Fanuc TP program (LS listing): UP021.LS

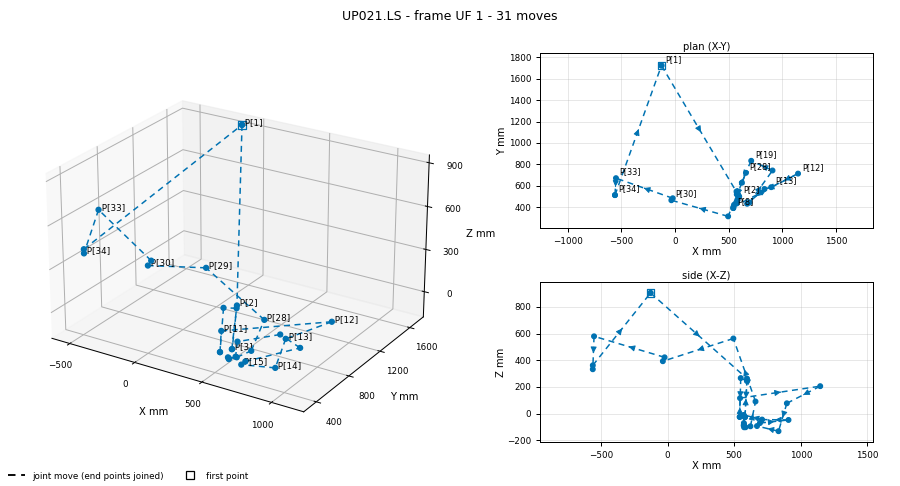
[picture p0: tool path of UP021.LS in frame UF 1, 31 of 37 moves have a stored position in this frame; points joined in program order, loops and branches not executed]
/PROG  UP021
/ATTR
OWNER		= GME;
COMMENT		= "Soldar en ST160i";
PROG_SIZE	= 14572;
CREATE		= DATE 03-01-31  TIME 09:09:48;
MODIFIED	= DATE 24-06-01  TIME 09:33:14;
FILE_NAME	= UP021;
VERSION		= 0;
LINE_COUNT	= 63;
MEMORY_SIZE	= 28492;
PROTECT		= READ_WRITE;
TCD:  STACK_SIZE	= 500,
      TASK_PRIORITY	= 50,
      TIME_SLICE	= 0,
      BUSY_LAMP_OFF	= 0,
      ABORT_REQUEST	= 0,
      PAUSE_REQUEST	= 0;
DEFAULT_GROUP	= 1,1,1,1,*;
CONTROL_CODE	= 00000000 00000000;
/APPL
/MN
   1:  UFRAME_NUM=1 ;
   2:  UTOOL_NUM=1 ;
   3:  PAYLOAD[1] ;
   4:  !Apagar Perfil Lib. 80 vs ST1600 ;
   5:  !Apagar Perfil Lib. 79 vs ST1600 ;
   6:  !Endender Anticol. 1 vs 1550R01 ;
   7:  !Endender Anticol. 3 vs 1610R01 ;
   8:J P[1] 100% CNT0 ACC100 TB    0.00sec,P-SPS    ;
      1:  TC_ONLINE (ON) ;
      2:  DO[23]=OFF ;
      3:  TIMER[3]=RESET ;
      4:  TIMER[3]=START ;
      5:  CALL MAKRO050    ;
      6:  !Lib. de Herramientas ;
      7:  DO[79]=ON ;
      8:  DO[80]=ON ;
      9:  !Lib. de Anticolisiones ;
     10:  DO[41]=ON ;
     11:  DO[42]=ON ;
     12:  DO[43]=ON ;
     13:  DO[44]=ON ;
     14:  !Apagar Pos. Base ;
     15:  DO[15]=OFF ;
     16:  !Robot en Trayectoria ;
     17:  DO[16]=ON ;
     18:  WAIT (DI[79] AND DI[80])    ;
     19:  DO[80]=OFF ;
     20:  DO[79]=OFF ;
     21:  !Encender Anticolisiones ;
     22:  DO[81]=ON ;
     23:  DO[83]=ON ;
     24:  CALL MAKRO020    ;
     25:  WAIT (DI[23])    ;
     26:  DO[23]=ON ;
     27:  TC_ONLINE (DI[41] AND DI[43] AND DI[79] AND DI[80] AND M[30] AND M[95]) ;
       ------ ;
   9:J P[2] 100% CNT100 ACC100 TB   0.00sec,P-SPS    ;
      1:  TC_ONLINE (DI[41] AND DI[43] AND DI[79] AND DI[80] AND M[30] AND M[95]) ;
       ------ ;
  10:J P[3] 100% CNT100 ACC100 TB   0.00sec,P-SPS    ;
      1:  TC_ONLINE (DI[41] AND DI[43] AND DI[79] AND DI[80] AND M[30] AND M[95]) ;
       ------ ;
  11:  !Punto de Sol. No. 11634 ;
  12:  !5qa803091b_p0008_h0210005900 ;
  13:J P[4] 100% CNT0 ACC100 TB    .10sec,P-SPS Tool_Offset,PR[11] Offset,PR[12]    ;
      1:  TC_ONLINE (ON) ;
      2:  DO[23]=OFF ;
      3:  WAIT (!DI[16] AND DI[23])    ;
      4:  CALL VW_USER(Basic1,EZSP,Nr1,ProgNr=99, , ,S-Punkt=11634,Fzg_Typ=7,EIN/AUS=ON) ;
      5:  GO[2]=(R[197]-2) ;
      6:  WAIT (!DI[129] OR DI[26])    ;
      7:  CALL MAKRO080    ;
      8:  WAIT (DI[23])    ;
      9:  DO[23]=ON ;
     10:  TC_ONLINE (DI[41] AND DI[43] AND DI[79] AND DI[80] AND M[30] AND M[95]) ;
       ------ ;
  14:J P[5] 100% CNT100 ACC100 TB   0.00sec,P-SPS    ;
      1:  TC_ONLINE (DI[41] AND DI[43] AND DI[79] AND DI[80] AND M[30] AND M[95]) ;
       ------ ;
  15:J P[6] 100% CNT100 ACC100 TB   0.00sec,P-SPS    ;
      1:  TC_ONLINE (DI[41] AND DI[43] AND DI[79] AND DI[80] AND M[30] AND M[95]) ;
       ------ ;
  16:J P[7] 100% CNT100 ACC100 TB   0.00sec,P-SPS    ;
      1:  TC_ONLINE (DI[41] AND DI[43] AND DI[79] AND DI[80] AND M[30] AND M[95]) ;
       ------ ;
  17:J P[8] 100% CNT100 ACC100 TB   0.00sec,P-SPS    ;
      1:  TC_ONLINE (DI[41] AND DI[43] AND DI[79] AND DI[80] AND M[30] AND M[95]) ;
       ------ ;
  18:  !Punto de Sol. No. 11635 ;
  19:  !5qa803091b_p0008_h0210006400 ;
  20:J P[9] 100% CNT0 ACC100 TB    .10sec,P-SPS Tool_Offset,PR[11] Offset,PR[12]    ;
      1:  TC_ONLINE (ON) ;
      2:  DO[23]=OFF ;
      3:  WAIT (!DI[16] AND DI[23])    ;
      4:  CALL VW_USER(Basic1,EZSP,Nr1,ProgNr=99, , ,S-Punkt=11635,Fzg_Typ=7,EIN/AUS=ON) ;
      5:  GO[2]=(R[197]-2) ;
      6:  WAIT (!DI[129] OR DI[26])    ;
      7:  CALL MAKRO080    ;
      8:  WAIT (DI[23])    ;
      9:  DO[23]=ON ;
     10:  TC_ONLINE (DI[41] AND DI[43] AND DI[79] AND DI[80] AND M[30] AND M[95]) ;
       ------ ;
  21:J P[10] 100% CNT100 ACC100 TB   0.00sec,P-SPS    ;
      1:  TC_ONLINE (DI[41] AND DI[43] AND DI[79] AND DI[80] AND M[30] AND M[95]) ;
       ------ ;
  22:J P[11] 100% CNT100 ACC100 TB   0.00sec,P-SPS    ;
      1:  TC_ONLINE (DI[41] AND DI[43] AND DI[79] AND DI[80] AND M[30] AND M[95]) ;
       ------ ;
  23:J P[12] 100% CNT100 ACC100 TB   0.00sec,P-SPS    ;
      1:  TC_ONLINE (DI[41] AND DI[43] AND DI[79] AND DI[80] AND M[30] AND M[95]) ;
       ------ ;
  24:J P[13] 100% CNT100 ACC100 TB   0.00sec,P-SPS    ;
      1:  TC_ONLINE (DI[41] AND DI[43] AND DI[79] AND DI[80] AND M[30] AND M[95]) ;
       ------ ;
  25:J P[14] 100% CNT100 ACC100 TB   0.00sec,P-SPS    ;
      1:  TC_ONLINE (DI[41] AND DI[43] AND DI[79] AND DI[80] AND M[30] AND M[95]) ;
       ------ ;
  26:J P[15] 100% CNT100 ACC100 TB   0.00sec,P-SPS    ;
      1:  TC_ONLINE (DI[41] AND DI[43] AND DI[79] AND DI[80] AND M[30] AND M[95]) ;
       ------ ;
  27:  !Punto de Sol. No. 11636 ;
  28:  !5qa803091b_p0008_h0210007000 ;
  29:J P[16] 100% CNT0 ACC100 TB    .10sec,P-SPS Tool_Offset,PR[11] Offset,PR[12]    ;
      1:  TC_ONLINE (ON) ;
      2:  DO[23]=OFF ;
      3:  WAIT (!DI[16] AND DI[23])    ;
      4:  CALL VW_USER(Basic1,EZSP,Nr1,ProgNr=99, , ,S-Punkt=11636,Fzg_Typ=7,EIN/AUS=ON) ;
      5:  GO[2]=(R[197]+10) ;
      6:  WAIT (!DI[129] OR DI[26])    ;
      7:  CALL MAKRO080    ;
      8:  WAIT (DI[23])    ;
      9:  DO[23]=ON ;
     10:  TC_ONLINE (DI[41] AND DI[43] AND DI[79] AND DI[80] AND M[30] AND M[95]) ;
       ------ ;
  30:J P[17] 100% CNT100 ACC100 TB   0.00sec,P-SPS    ;
      1:  TC_ONLINE (DI[41] AND DI[43] AND DI[79] AND DI[80] AND M[30] AND M[95]) ;
       ------ ;
  31:J P[18] 100% CNT100 ACC100 TB   0.00sec,P-SPS    ;
      1:  TC_ONLINE (DI[41] AND DI[43] AND DI[79] AND DI[80] AND M[30] AND M[95]) ;
       ------ ;
  32:J P[19] 100% CNT100 ACC100 TB   0.00sec,P-SPS    ;
      1:  TC_ONLINE (DI[41] AND DI[43] AND DI[79] AND DI[80] AND M[30] AND M[95]) ;
       ------ ;
  33:J P[20] 100% CNT100 ACC100 TB   0.00sec,P-SPS    ;
      1:  TC_ONLINE (DI[41] AND DI[43] AND DI[79] AND DI[80] AND M[30] AND M[95]) ;
       ------ ;
  34:J P[21] 100% CNT100 ACC100 TB   0.00sec,P-SPS    ;
      1:  TC_ONLINE (DI[41] AND DI[43] AND DI[79] AND DI[80] AND M[30] AND M[95]) ;
       ------ ;
  35:J P[22] 100% CNT100 ACC100 TB   0.00sec,P-SPS    ;
      1:  TC_ONLINE (DI[41] AND DI[43] AND DI[79] AND DI[80] AND M[30] AND M[95]) ;
       ------ ;
  36:J P[23] 100% CNT100 ACC100 TB   0.00sec,P-SPS    ;
      1:  TC_ONLINE (DI[41] AND DI[43] AND DI[79] AND DI[80] AND M[30] AND M[95]) ;
       ------ ;
  37:  !Punto de Sol. No. 11637 ;
  38:  !5qa803091b_p0008_h0210006100 ;
  39:J P[24] 100% CNT0 ACC100 TB    .10sec,P-SPS Tool_Offset,PR[11] Offset,PR[12]    ;
      1:  TC_ONLINE (ON) ;
      2:  DO[23]=OFF ;
      3:  WAIT (!DI[16] AND DI[23])    ;
      4:  CALL VW_USER(Basic1,EZSP,Nr1,ProgNr=99, , ,S-Punkt=11637,Fzg_Typ=7,EIN/AUS=ON) ;
      5:  GO[2]=(R[197]+10) ;
      6:  WAIT (!DI[129] OR DI[26])    ;
      7:  CALL MAKRO080    ;
      8:  WAIT (DI[23])    ;
      9:  DO[23]=ON ;
     10:  TC_ONLINE (DI[41] AND DI[43] AND DI[79] AND DI[80] AND M[30] AND M[95]) ;
       ------ ;
  40:J P[25] 100% CNT100 ACC100 TB   0.00sec,P-SPS    ;
      1:  TC_ONLINE (DI[41] AND DI[43] AND DI[79] AND DI[80] AND M[30] AND M[95]) ;
       ------ ;
  41:J P[26] 100% CNT100 ACC100 TB   0.00sec,P-SPS    ;
      1:  TC_ONLINE (DI[41] AND DI[43] AND DI[79] AND DI[80] AND M[30] AND M[95]) ;
       ------ ;
  42:J P[27] 100% CNT100 ACC100 TB   0.00sec,P-SPS    ;
      1:  TC_ONLINE (DI[41] AND DI[43] AND DI[79] AND DI[80] AND M[30] AND M[95]) ;
       ------ ;
  43:J P[28] 100% CNT100 ACC100 TB   0.00sec,P-SPS    ;
      1:  TC_ONLINE (DI[41] AND DI[43] AND DI[79] AND DI[80] AND M[30] AND M[95]) ;
       ------ ;
  44:J P[29] 100% CNT100 ACC100 TB   0.00sec,P-SPS    ;
      1:  TC_ONLINE (DI[41] AND DI[43] AND DI[79] AND DI[80] AND M[30] AND M[95]) ;
       ------ ;
  45:J P[30] 100% CNT100 ACC100 TB   0.00sec,P-SPS    ;
      1:  TC_ONLINE (DI[41] AND DI[43] AND DI[79] AND DI[80] AND M[30] AND M[95]) ;
       ------ ;
  46:  !no soldar CKD ;
  47:  !Punto de Sol. No. 11638 ;
  48:  !5qa802035b_018_sps0033_R ;
  49:J P[31] 100% CNT0 ACC100 TB    .10sec,P-SPS Tool_Offset,PR[11] Offset,PR[12]    ;
      1:  TC_ONLINE (ON) ;
      2:  DO[23]=OFF ;
      3:  WAIT (!DI[16] AND DI[23])    ;
      4:  CALL VW_USER(Basic1,EZSP,Nr1,ProgNr=99, , ,S-Punkt=11638,Fzg_Typ=7,EIN/AUS=ON) ;
      5:  GO[2]=(R[197]-4) ;
      6:  WAIT (!DI[129] OR DI[26])    ;
      7:  CALL MAKRO080    ;
      8:  WAIT (DI[23])    ;
      9:  DO[23]=ON ;
     10:  TC_ONLINE (DI[41] AND DI[43] AND DI[79] AND DI[80] AND M[30] AND M[95]) ;
       ------ ;
  50:J P[32] 100% CNT100 ACC100 TB   0.00sec,P-SPS    ;
      1:  TC_ONLINE (DI[41] AND DI[43] AND DI[79] AND DI[80] AND M[30] AND M[95]) ;
       ------ ;
  51:J P[33] 100% FINE ACC100 DB    0.0mm,P-SPS    ;
      1:  TC_ONLINE (DI[41] AND DI[43] AND DI[79] AND DI[80] AND M[30] AND M[95]) ;
       ------ ;
  52:J P[34] 100% CNT100 ACC100 TB   0.00sec,P-SPS    ;
      1:  TC_ONLINE (DI[41] AND DI[43] AND DI[79] AND DI[80] AND M[30] AND M[95]) ;
       ------ ;
  53:  !no soldar CKD ;
  54:  !Punto de Sol. No. 11639 ;
  55:  !Fin de Trabajo 1 ;
  56:  !5qa802035b_018_sps0021_R ;
  57:J P[35] 100% CNT0 ACC100 TB    0.00sec,P-SPS Tool_Offset,PR[11] Offset,PR[12]    ;
      1:  TC_ONLINE (ON) ;
      2:  DO[23]=OFF ;
      3:  WAIT (!DI[16] AND DI[23])    ;
      4:  CALL VW_USER(Basic1,EZSP,Nr1,ProgNr=99, , ,S-Punkt=11639,Fzg_Typ=7,EIN/AUS=ON) ;
      5:  GO[2]=(R[197]) ;
      6:  WAIT (!DI[129] OR DI[26])    ;
      7:  CALL MAKRO080    ;
      8:  IF (!DI[145] AND !DI[129]),CALL MAKRO001 ;
      9:  WAIT (DI[23])    ;
     10:  DO[23]=ON ;
     11:  TC_ONLINE (DI[41] AND DI[43] AND DI[79] AND DI[80] AND M[30] AND M[95]) ;
       ------ ;
  58:J P[36] 100% CNT100 ACC100 TB   0.00sec,P-SPS    ;
      1:  TC_ONLINE (DI[41] AND DI[43] AND DI[79] AND DI[80] AND M[30] AND M[95]) ;
       ------ ;
  59:  !Encender Perfil Lib 80 vs ST1600 ;
  60:  !Encender Perfil Lib 79 vs ST1600 ;
  61:  !Apagar Anticol. 1 vs 1550R01 ;
  62:  !Apagar Anticol. 3 vs 1610R01 ;
  63:J P[37] 100% CNT0 ACC100 TB    .10sec,P-SPS    ;
      1:  TC_ONLINE (ON) ;
      2:  DO[23]=OFF ;
      3:  TIMER[3]=STOP ;
      4:  DO[41]=ON ;
      5:  DO[43]=ON ;
      6:  DO[79]=ON ;
      7:  DO[80]=ON ;
      8:  WAIT (DI[23])    ;
      9:  DO[23]=ON ;
     10:  TC_ONLINE (M[30] AND M[95]) ;
       ------ ;
/POS
P[1]{
   GP1:
	UF : 1, UT : 1,		CONFIG : 'N U T, 0, 0, 0',
	X =  -127.542  mm,	Y =  1721.879  mm,	Z =   904.497  mm,
	W =  -170.302 deg,	P =     1.120 deg,	R =   132.757 deg
   GP2:
	UF : 1, UT : 1,
	J1=   100.000  mm
   GP3:
	UF : 1, UT : 1,
	J1=     0.000  mm
   GP4:
	UF : 1, UT : 1,
	J1=     0.000  mm
};
P[2]{
   GP1:
	UF : 1, UT : 1,		CONFIG : 'N U T, 0, 0, 0',
	X =   596.207  mm,	Y =   502.707  mm,	Z =   261.856  mm,
	W =  -176.468 deg,	P =     7.977 deg,	R =    93.412 deg
   GP2:
	UF : 1, UT : 1,
	J1=   125.000  mm
   GP3:
	UF : 1, UT : 1,
	J1=     0.000  mm
   GP4:
	UF : 1, UT : 1,
	J1=     0.000  mm
};
P[3]{
   GP1:
	UF : 1, UT : 1,		CONFIG : 'N U T, 0, 0, 0',
	X =   580.717  mm,	Y =   471.716  mm,	Z =   -27.286  mm,
	W =  -176.468 deg,	P =     7.977 deg,	R =    93.413 deg
   GP2:
	UF : 1, UT : 1,
	J1=   125.000  mm
   GP3:
	UF : 1, UT : 1,
	J1=     0.000  mm
   GP4:
	UF : 1, UT : 1,
	J1=     0.000  mm
};
P[4]{
   GP1:
	UF : 1, UT : 1,		CONFIG : 'N U T, 0, 0, 0',
	X =   579.173  mm,	Y =   480.025  mm,	Z =   -30.338  mm,
	W =  -175.927 deg,	P =     7.716 deg,	R =    97.374 deg
   GP2:
	UF : 1, UT : 1,
	J1=    14.100  mm
   GP3:
	UF : 1, UT : 1,
	J1=     0.000  mm
   GP4:
	UF : 1, UT : 1,
	J1=     0.000  mm
};
P[5]{
   GP1:
	UF : 1, UT : 1,		CONFIG : 'N U T, 0, 0, 0',
	X =   581.000  mm,	Y =   466.971  mm,	Z =   -26.620  mm,
	W =  -176.468 deg,	P =     7.977 deg,	R =    93.413 deg
   GP2:
	UF : 1, UT : 1,
	J1=   125.000  mm
   GP3:
	UF : 1, UT : 1,
	J1=     0.000  mm
   GP4:
	UF : 1, UT : 1,
	J1=     0.000  mm
};
P[6]{
   GP1:
	UF : 1, UT : 1,		CONFIG : 'N U T, 0, 0, 0',
	X =   595.238  mm,	Y =   500.117  mm,	Z =   243.816  mm,
	W =  -176.468 deg,	P =     7.977 deg,	R =    93.412 deg
   GP2:
	UF : 1, UT : 1,
	J1=   125.000  mm
   GP3:
	UF : 1, UT : 1,
	J1=     0.000  mm
   GP4:
	UF : 1, UT : 1,
	J1=     0.000  mm
};
P[7]{
   GP1:
	UF : 1, UT : 1,		CONFIG : 'N U T, 0, 0, 0',
	X =   548.949  mm,	Y =   423.931  mm,	Z =   265.870  mm,
	W =   176.635 deg,	P =    -4.508 deg,	R =   -86.117 deg
   GP2:
	UF : 1, UT : 1,
	J1=   123.300  mm
   GP3:
	UF : 1, UT : 1,
	J1=     0.000  mm
   GP4:
	UF : 1, UT : 1,
	J1=     0.000  mm
};
P[8]{
   GP1:
	UF : 1, UT : 1,		CONFIG : 'N U T, 0, 0, 0',
	X =   541.543  mm,	Y =   393.353  mm,	Z =   -25.633  mm,
	W =   178.696 deg,	P =     7.978 deg,	R =   -86.999 deg
   GP2:
	UF : 1, UT : 1,
	J1=   184.230  mm
   GP3:
	UF : 1, UT : 1,
	J1=     0.000  mm
   GP4:
	UF : 1, UT : 1,
	J1=     0.000  mm
};
P[9]{
   GP1:
	UF : 1, UT : 1,		CONFIG : 'N U T, 0, 0, 0',
	X =   535.657  mm,	Y =   384.383  mm,	Z =   -21.270  mm,
	W =   178.700 deg,	P =     7.998 deg,	R =   -87.000 deg
   GP2:
	UF : 1, UT : 1,
	J1=    21.214  mm
   GP3:
	UF : 1, UT : 1,
	J1=     0.000  mm
   GP4:
	UF : 1, UT : 1,
	J1=     0.000  mm
};
P[10]{
   GP1:
	UF : 1, UT : 1,		CONFIG : 'N U T, 0, 0, 0',
	X =   541.543  mm,	Y =   393.353  mm,	Z =   -25.633  mm,
	W =   178.696 deg,	P =     7.978 deg,	R =   -86.999 deg
   GP2:
	UF : 1, UT : 1,
	J1=   184.230  mm
   GP3:
	UF : 1, UT : 1,
	J1=     0.000  mm
   GP4:
	UF : 1, UT : 1,
	J1=     0.000  mm
};
P[11]{
   GP1:
	UF : 1, UT : 1,		CONFIG : 'N U T, 0, 0, 0',
	X =   543.886  mm,	Y =   405.233  mm,	Z =   115.349  mm,
	W =   178.700 deg,	P =     8.003 deg,	R =   -87.001 deg
   GP2:
	UF : 1, UT : 1,
	J1=   195.035  mm
   GP3:
	UF : 1, UT : 1,
	J1=     0.000  mm
   GP4:
	UF : 1, UT : 1,
	J1=     0.000  mm
};
P[12]{
   GP1:
	UF : 1, UT : 1,		CONFIG : 'N U T, 0, 0, 0',
	X =  1145.296  mm,	Y =   714.799  mm,	Z =   205.075  mm,
	W =   175.360 deg,	P =   -36.825 deg,	R =  -109.073 deg
   GP2:
	UF : 1, UT : 1,
	J1=   125.000  mm
   GP3:
	UF : 1, UT : 1,
	J1=     0.000  mm
   GP4:
	UF : 1, UT : 1,
	J1=     0.000  mm
};
P[13]{
   GP1:
	UF : 1, UT : 1,		CONFIG : 'N U T, 0, 0, 0',
	X =   895.080  mm,	Y =   588.023  mm,	Z =    76.712  mm,
	W =   154.499 deg,	P =   -66.911 deg,	R =  -110.430 deg
   GP2:
	UF : 1, UT : 1,
	J1=   124.497  mm
   GP3:
	UF : 1, UT : 1,
	J1=     0.000  mm
   GP4:
	UF : 1, UT : 1,
	J1=     0.000  mm
};
P[14]{
   GP1:
	UF : 1, UT : 1,		CONFIG : 'N U T, 0, 0, 0',
	X =   832.340  mm,	Y =   571.049  mm,	Z =  -132.697  mm,
	W =  -179.033 deg,	P =   -75.571 deg,	R =  -137.274 deg
   GP2:
	UF : 1, UT : 1,
	J1=   160.000  mm
   GP3:
	UF : 1, UT : 1,
	J1=     0.000  mm
   GP4:
	UF : 1, UT : 1,
	J1=     0.000  mm
};
P[15]{
   GP1:
	UF : 1, UT : 1,		CONFIG : 'N U T, 0, 0, 0',
	X =   671.028  mm,	Y =   433.463  mm,	Z =   -94.035  mm,
	W =  -163.603 deg,	P =   -85.208 deg,	R =  -151.224 deg
   GP2:
	UF : 1, UT : 1,
	J1=   140.000  mm
   GP3:
	UF : 1, UT : 1,
	J1=     0.000  mm
   GP4:
	UF : 1, UT : 1,
	J1=     0.000  mm
};
P[16]{
   GP1:
	UF : 1, UT : 1,		CONFIG : 'N U T, 0, 0, 0',
	X =   663.425  mm,	Y =   425.299  mm,	Z =   -53.189  mm,
	W =  -143.117 deg,	P =   -88.278 deg,	R =  -170.993 deg
   GP2:
	UF : 1, UT : 1,
	J1=    26.100  mm
   GP3:
	UF : 1, UT : 1,
	J1=     0.000  mm
   GP4:
	UF : 1, UT : 1,
	J1=     0.000  mm
};
P[17]{
   GP1:
	UF : 1, UT : 1,		CONFIG : 'N U T, 0, 0, 0',
	X =   693.231  mm,	Y =   444.844  mm,	Z =   -71.614  mm,
	W =     3.860 deg,	P =   -88.327 deg,	R =    44.457 deg
   GP2:
	UF : 1, UT : 1,
	J1=   123.386  mm
   GP3:
	UF : 1, UT : 1,
	J1=     0.000  mm
   GP4:
	UF : 1, UT : 1,
	J1=     0.000  mm
};
P[18]{
   GP1:
	UF : 1, UT : 1,		CONFIG : 'N U T, 0, 0, 0',
	X =   907.349  mm,	Y =   743.785  mm,	Z =   -48.294  mm,
	W =   179.443 deg,	P =   -77.707 deg,	R =  -131.143 deg
   GP2:
	UF : 1, UT : 1,
	J1=   200.000  mm
   GP3:
	UF : 1, UT : 1,
	J1=     0.000  mm
   GP4:
	UF : 1, UT : 1,
	J1=     0.000  mm
};
P[19]{
   GP1:
	UF : 1, UT : 1,		CONFIG : 'N U T, 0, 0, 0',
	X =   708.992  mm,	Y =   833.948  mm,	Z =   -45.348  mm,
	W =   174.604 deg,	P =   -72.662 deg,	R =  -121.135 deg
   GP2:
	UF : 1, UT : 1,
	J1=   189.300  mm
   GP3:
	UF : 1, UT : 1,
	J1=     0.000  mm
   GP4:
	UF : 1, UT : 1,
	J1=     0.000  mm
};
P[20]{
   GP1:
	UF : 1, UT : 1,		CONFIG : 'N U T, 0, 0, 0',
	X =   571.724  mm,	Y =   547.931  mm,	Z =   -10.847  mm,
	W =   148.202 deg,	P =   -86.004 deg,	R =   -84.037 deg
   GP2:
	UF : 1, UT : 1,
	J1=   189.300  mm
   GP3:
	UF : 1, UT : 1,
	J1=     0.000  mm
   GP4:
	UF : 1, UT : 1,
	J1=     0.000  mm
};
P[21]{
   GP1:
	UF : 1, UT : 1,		CONFIG : 'N U T, 0, 0, -1',
	X =   574.306  mm,	Y =   521.337  mm,	Z =  -103.269  mm,
	W =  -164.049 deg,	P =   -86.313 deg,	R =  -124.103 deg
   GP2:
	UF : 1, UT : 1,
	J1=   189.300  mm
   GP3:
	UF : 1, UT : 1,
	J1=     0.000  mm
   GP4:
	UF : 1, UT : 1,
	J1=     0.000  mm
};
P[22]{
   GP1:
	UF : 1, UT : 1,		CONFIG : 'N U T, 0, 0, -1',
	X =   570.874  mm,	Y =   448.514  mm,	Z =   -89.375  mm,
	W =   -28.476 deg,	P =   -88.160 deg,	R =   107.064 deg
   GP2:
	UF : 1, UT : 1,
	J1=   146.387  mm
   GP3:
	UF : 1, UT : 1,
	J1=     0.000  mm
   GP4:
	UF : 1, UT : 1,
	J1=     0.000  mm
};
P[23]{
   GP1:
	UF : 1, UT : 1,		CONFIG : 'N U T, 0, 0, -1',
	X =   572.485  mm,	Y =   436.058  mm,	Z =   -71.706  mm,
	W =    -3.346 deg,	P =   -87.918 deg,	R =    86.155 deg
   GP2:
	UF : 1, UT : 1,
	J1=    67.043  mm
   GP3:
	UF : 1, UT : 1,
	J1=     0.000  mm
   GP4:
	UF : 1, UT : 1,
	J1=     0.000  mm
};
P[24]{
   GP1:
	UF : 1, UT : 1,		CONFIG : 'N U T, 0, 1, 0',
	X =   591.997  mm,	Y =   444.102  mm,	Z =   -58.846  mm,
	W =     9.794 deg,	P =   -87.982 deg,	R =    82.383 deg
   GP2:
	UF : 1, UT : 1,
	J1=    30.000  mm
   GP3:
	UF : 1, UT : 1,
	J1=     0.000  mm
   GP4:
	UF : 1, UT : 1,
	J1=     0.000  mm
};
P[25]{
   GP1:
	UF : 1, UT : 1,		CONFIG : 'N U T, 0, 0, -1',
	X =   573.364  mm,	Y =   444.944  mm,	Z =   -81.600  mm,
	W =  -160.763 deg,	P =   -89.630 deg,	R =  -116.426 deg
   GP2:
	UF : 1, UT : 1,
	J1=   129.157  mm
   GP3:
	UF : 1, UT : 1,
	J1=     0.000  mm
   GP4:
	UF : 1, UT : 1,
	J1=     0.000  mm
};
P[26]{
   GP1:
	UF : 1, UT : 1,		CONFIG : 'N U T, 0, 0, -1',
	X =   585.119  mm,	Y =   517.785  mm,	Z =  -103.069  mm,
	W =  -164.048 deg,	P =   -86.313 deg,	R =  -124.103 deg
   GP2:
	UF : 1, UT : 1,
	J1=   189.300  mm
   GP3:
	UF : 1, UT : 1,
	J1=     0.000  mm
   GP4:
	UF : 1, UT : 1,
	J1=     0.000  mm
};
P[27]{
   GP1:
	UF : 1, UT : 1,		CONFIG : 'N U T, 0, 0, 0',
	X =   621.794  mm,	Y =   629.533  mm,	Z =   -95.964  mm,
	W =  -176.641 deg,	P =   -72.546 deg,	R =  -111.380 deg
   GP2:
	UF : 1, UT : 1,
	J1=   189.200  mm
   GP3:
	UF : 1, UT : 1,
	J1=     0.000  mm
   GP4:
	UF : 1, UT : 1,
	J1=     0.000  mm
};
P[28]{
   GP1:
	UF : 1, UT : 1,		CONFIG : 'N U T, 0, 0, 0',
	X =   659.865  mm,	Y =   721.962  mm,	Z =    90.033  mm,
	W =   175.247 deg,	P =   -63.696 deg,	R =  -111.510 deg
   GP2:
	UF : 1, UT : 1,
	J1=   189.300  mm
   GP3:
	UF : 1, UT : 1,
	J1=     0.000  mm
   GP4:
	UF : 1, UT : 1,
	J1=     0.000  mm
};
P[29]{
   GP1:
	UF : 1, UT : 1,		CONFIG : 'N U T, 0, 0, 0',
	X =   493.795  mm,	Y =   316.297  mm,	Z =   562.676  mm,
	W =  -163.963 deg,	P =   -49.377 deg,	R =  -123.525 deg
   GP2:
	UF : 1, UT : 1,
	J1=    80.000  mm
   GP3:
	UF : 1, UT : 1,
	J1=     0.000  mm
   GP4:
	UF : 1, UT : 1,
	J1=     0.000  mm
};
P[30]{
   GP1:
	UF : 1, UT : 1,		CONFIG : 'N U T, 0, 0, -1',
	X =   -35.265  mm,	Y =   466.444  mm,	Z =   392.223  mm,
	W =  -165.513 deg,	P =    14.948 deg,	R =    76.257 deg
   GP2:
	UF : 1, UT : 1,
	J1=   125.000  mm
   GP3:
	UF : 1, UT : 1,
	J1=     0.000  mm
   GP4:
	UF : 1, UT : 1,
	J1=     0.000  mm
};
P[31]{
   GP1:
	UF : 1, UT : 1,		CONFIG : 'N U T, 0, 0, -1',
	X =   -39.123  mm,	Y =   480.360  mm,	Z =   284.124  mm,
	W =  -165.563 deg,	P =    14.928 deg,	R =    76.062 deg
   GP2:
	UF : 1, UT : 1,
	J1=    30.000  mm
   GP3:
	UF : 1, UT : 1,
	J1=     0.000  mm
   GP4:
	UF : 1, UT : 1,
	J1=     0.000  mm
};
P[32]{
   GP1:
	UF : 1, UT : 1,		CONFIG : 'N U T, 0, 0, -1',
	X =   -22.267  mm,	Y =   485.036  mm,	Z =   421.540  mm,
	W =  -165.513 deg,	P =    14.944 deg,	R =    76.259 deg
   GP2:
	UF : 1, UT : 1,
	J1=    80.000  mm
   GP3:
	UF : 1, UT : 1,
	J1=     0.000  mm
   GP4:
	UF : 1, UT : 1,
	J1=     0.000  mm
};
P[33]{
   GP1:
	UF : 1, UT : 1,		CONFIG : 'N U T, 0, 0, 0',
	X =  -551.441  mm,	Y =   672.230  mm,	Z =   579.194  mm,
	W =  -157.989 deg,	P =     3.152 deg,	R =    74.028 deg
   GP2:
	UF : 1, UT : 1,
	J1=   100.000  mm
   GP3:
	UF : 1, UT : 1,
	J1=     0.000  mm
   GP4:
	UF : 1, UT : 1,
	J1=     0.000  mm
};
P[34]{
   GP1:
	UF : 1, UT : 1,		CONFIG : 'N U T, 0, 0, 0',
	X =  -560.866  mm,	Y =   514.351  mm,	Z =   332.029  mm,
	W =  -153.408 deg,	P =     -.686 deg,	R =    89.026 deg
   GP2:
	UF : 1, UT : 1,
	J1=    61.600  mm
   GP3:
	UF : 1, UT : 1,
	J1=     0.000  mm
   GP4:
	UF : 1, UT : 1,
	J1=     0.000  mm
};
P[35]{
   GP1:
	UF : 1, UT : 1,		CONFIG : 'N U T, 0, 0, 0',
	X =  -578.531  mm,	Y =   523.822  mm,	Z =   297.986  mm,
	W =  -163.790 deg,	P =    -3.677 deg,	R =    89.851 deg
   GP2:
	UF : 1, UT : 1,
	J1=    13.700  mm
   GP3:
	UF : 1, UT : 1,
	J1=     0.000  mm
   GP4:
	UF : 1, UT : 1,
	J1=     0.000  mm
};
P[36]{
   GP1:
	UF : 1, UT : 1,		CONFIG : 'N U T, 0, 0, 0',
	X =  -560.713  mm,	Y =   514.070  mm,	Z =   361.307  mm,
	W =  -153.408 deg,	P =     -.686 deg,	R =    89.026 deg
   GP2:
	UF : 1, UT : 1,
	J1=    61.600  mm
   GP3:
	UF : 1, UT : 1,
	J1=     0.000  mm
   GP4:
	UF : 1, UT : 1,
	J1=     0.000  mm
};
P[37]{
   GP1:
	UF : 1, UT : 1,		CONFIG : 'N U T, 0, 0, 0',
	X =  -127.542  mm,	Y =  1721.879  mm,	Z =   904.497  mm,
	W =  -170.302 deg,	P =     1.120 deg,	R =   132.757 deg
   GP2:
	UF : 1, UT : 1,
	J1=   100.000  mm
   GP3:
	UF : 1, UT : 1,
	J1=     0.000  mm
   GP4:
	UF : 1, UT : 1,
	J1=     0.000  mm
};
/END
